Staubli VAL3: setIOTask.pgx

program setIOTask()
  local point l_pHere
  local point l_pPrev
  local num l_nNum
begin
  l_pPrev=here(tTool,FrmDraw)
  l_nNum=0
  while true
    if bSetIO==true
      l_pHere=here(tTool,FrmDraw)
      if distance(l_pPrev,l_pHere)>=1
        //        io:fOut0=false
        //        delay(0)
        //        io:fOut0=true
        l_pPrev=l_pHere
        l_nNum=l_nNum+1
        nIONum=l_nNum
        //        gotoxy(35,11)
        //        put(nIONum)
      endIf
    endIf
    gotoxy(35,11)
    put(nTime)
    delay(0.1)
  endWhile
end
